Fanuc TP program (LS listing): S107_PK_T13N70.LS

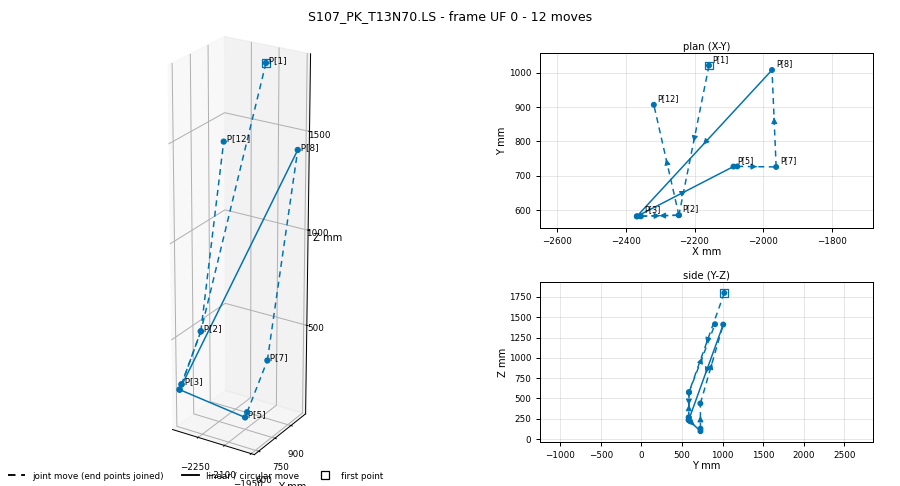
[picture p0: tool path of S107_PK_T13N70.LS in frame UF 0, 12 of 12 moves have a stored position in this frame; points joined in program order, loops and branches not executed]
/PROG  S107_PK_T13N70
/ATTR
OWNER		= MNEDITOR;
COMMENT		= "TL PCK TYP1 N70";
PROG_SIZE	= 4376;
CREATE		= DATE 21-06-09  TIME 09:54:06;
MODIFIED	= DATE 21-06-09  TIME 12:46:12;
FILE_NAME	= S107_PK_;
VERSION		= 0;
LINE_COUNT	= 155;
MEMORY_SIZE	= 4796;
PROTECT		= READ_WRITE;
STORAGE		= SHADOW;
TCD:  STACK_SIZE	= 0,
      TASK_PRIORITY	= 50,
      TIME_SLICE	= 0,
      BUSY_LAMP_OFF	= 0,
      ABORT_REQUEST	= 0,
      PAUSE_REQUEST	= 0;
DEFAULT_GROUP	= 1,*,*,*,*;
CONTROL_CODE	= 00000000 00000000;
/APPL
  HANDLING : TRUE ;
/MN
   1:  !******************************** ;
   2:  ! PATH - PK TOOL FROM N3=STA 70 ;
   3:  !******************************** ;
   4:  !* Robot ID: XXXXXR02B1 ;
   5:  !*    F-19XXXX ;
   6:  !* Line: XXXXXXXX ;
   7:  !* Platform: XX ;
   8:  !* Tool ID: TOOL xx ;
   9:  !* Program: S002_PK_TxxN3_R02 ;
  10:  !* Application: TOOL PICK ;
  11:  !******************************** ;
  12:  ! Author- Esys Automation ;
  13:  !******************************** ;
  14:   ;
  15:  !++++++++++++++++++++++++++++++++ ;
  16:  !ASSIGN PROGRAM PATH VALUES ;
  17:  !-------------------------------- ;
  18:  !Set ATI Tool and World UFrame ;
  19:  UTOOL_NUM=14 ;
  20:  UFRAME_NUM=0 ;
  21:  !++++++++++++++++++++++++++++++++ ;
  22:   ;
  23:  !******************************** ;
  24:  !BEGINNING OF PROGRAM PATH ;
  25:  !MOVE TO NEST 3 TOOL PICK ;
  26:  !******************************** ;
  27:   ;
  28:  !-------------------------------- ;
  29:  LBL[10:MOVE TO TL PICK] ;
  30:   ;
  31:  SET SEGMENT(52) ;
  32:  !SEG(52), Approach Tool Pick ;
  33:   ;
  34:J P[1] 100% CNT100    ;
  35:J P[2] 100% CNT100    ;
  36:J P[3] 100% CNT100    ;
  37:   ;
  38:L P[4:Pick Tool] 50mm/sec FINE    ;
  39:   ;
  40:  !-------------------------------- ;
  41:  LBL[20:LATCH TOOL] ;
  42:  LATCH TOOL    ;
  43:   ;
  44:  Set MH Tool(4) ;
  45:  Release Part(5) ;
  46:  VACUUM CAN 1 OFF(6,7) ;
  47:   ;
  48:  !Add MH Ethernet Device from ;
  49:  !I/O Ethernet table ;
  50:  !which tool has ;
  51:   ;
  52:  !ADD DEVICE ONLINE CALLS ;
  53:  !WITHOUT STATUS CHECK ARG ;
  54:  !FOR ALL EOAT DEVICES ;
  55:  !CALL EN_ONLN(x,y) ;
  56:  !x = EOAT ENET Node # ;
  57:  !y = wait time ;
  58:  CALL EN_ONLN(31,5) ;
  59:  CALL EN_AROFF(31) ;
  60:   ;
  61:  !If TL LCH Pass, Return Home ;
  62:  !If TL LCH Fail, Unlatch TL, ;
  63:  !  MHFault, and Return Home ;
  64:  IF R[170]=1,JMP LBL[30] ;
  65:   ;
  66:  SELECT R[168]=6,JMP LBL[80] ;
  67:         ELSE,JMP LBL[99] ;
  68:   ;
  69:  !-------------------------------- ;
  70:  LBL[30:TOOL CHECK] ;
  71:   ;
  72:  ! Check if Tool Match with PLC ;
  73:  CALL TL_CHK_KM(R[156]) ;
  74:   ;
  75:  !If TL CHK Pass, Return Home ;
  76:  !If TL CHK Fail, Unlatch Tool, ;
  77:  !  MHFault, and Return Home ;
  78:  IF R[170]=1,JMP LBL[40] ;
  79:  IF R[170]=0,JMP LBL[905] ;
  80:   ;
  81:  !-------------------------------- ;
  82:  LBL[40:COMPLETE PATH] ;
  83:  !TL PK COMPLETE. MOVE AWAY ;
  84:  !AND RETURN HOME ;
  85:   ;
  86:  !Set New Tool and World Frame ;
  87:  UTOOL_NUM=2 ;
  88:  UFRAME_NUM=0 ;
  89:   ;
  90:  !Set Payload= Tool ;
  91:  R[221]=2    ;
  92:  PAYLOAD[R[221]] ;
  93:   ;
  94:  SET SEGMENT(53) ;
  95:  !SEG(53), Tool Pick Depart ;
  96:   ;
  97:L P[5] 50mm/sec FINE    ;
  98:   ;
  99:L P[6] 1000mm/sec CNT100    ;
 100:J P[7] 100% CNT100    ;
 101:J P[8] 100% CNT100    ;
 102:   ;
 103:   ;
 104:  ! Move To Home ;
 105:  JMP LBL[100] ;
 106:   ;
 107:  !-------------------------------- ;
 108:  LBL[80:LATCHING FAULT] ;
 109:  !MOVE BACK TO HOME WITHOUT TOOL ;
 110:  !on Reverse Path before Tool Pick ;
 111:   ;
 112:  UNLATCH TOOL    ;
 113:   ;
 114:  UFRAME_NUM=0 ;
 115:  UTOOL_NUM=14 ;
 116:   ;
 117:L P[9] 50mm/sec FINE    ;
 118:   ;
 119:L P[10] 1000mm/sec CNT100    ;
 120:J P[11] 100% CNT100    ;
 121:J P[12] 100% CNT100    ;
 122:   ;
 123:   ;
 124:  SET SEGMENT(63) ;
 125:  !SEG(63), Robot Move to Home ;
 126:   ;
 127:  R[132]=0    ;
 128:  GO[71]=0 ;
 129:   ;
 130:  ! Move To Home ;
 131:  JMP LBL[100] ;
 132:   ;
 133:  !-------------------------------- ;
 134:  LBL[99:ABORT PROGRAM] ;
 135:  MESSAGE[...] ;
 136:  MESSAGE[ABORT PROGRAM] ;
 137:  ABORT ;
 138:   ;
 139:  !-------------------------------- ;
 140:  LBL[100:END OF PROGRAM] ;
 141:  END ;
 142:   ;
 143:  !***********FAULTS*********** ;
 144:  LBL[905:Invalid Tool Num] ;
 145:  MESSAGE[...] ;
 146:  MESSAGE[TOOL CHANGER FAULT] ;
 147:  MESSAGE[ ROBOT LATCHED TO] ;
 148:  MESSAGE[ WRONG TOOL.] ;
 149:  MESSAGE[ GI[70] DOES NOT ] ;
 150:  MESSAGE[ MATCH TOOL ID ] ;
 151:  DO[523]=ON ;
 152:  UALM[3] ;
 153:  DO[523]=OFF ;
 154:  JMP LBL[80] ;
 155:   ;
/POS
P[1]{
   GP1:
	UF : 0, UT : 14,		CONFIG : 'N U T, 0, 0, 0',
	X = -2157.965  mm,	Y =  1020.774  mm,	Z =  1799.157  mm,
	W =  -148.691 deg,	P =     -.556 deg,	R =    64.095 deg
};
P[2]{
   GP1:
	UF : 0, UT : 14,		CONFIG : 'N U T, 0, 0, 0',
	X = -2245.406  mm,	Y =   585.737  mm,	Z =   576.045  mm,
	W =  -160.449 deg,	P =      .486 deg,	R =    90.889 deg
};
P[3]{
   GP1:
	UF : 0, UT : 14,		CONFIG : 'N U T, 0, 0, 0',
	X = -2356.425  mm,	Y =   582.838  mm,	Z =   265.364  mm,
	W =  -160.444 deg,	P =      .210 deg,	R =    91.666 deg
};
P[4:"Pick Tool"]{
   GP1:
	UF : 0, UT : 14,		CONFIG : 'N U T, 0, 0, 0',
	X = -2367.590  mm,	Y =   582.398  mm,	Z =   233.916  mm,
	W =  -160.444 deg,	P =      .209 deg,	R =    91.666 deg
};
P[5]{
   GP1:
	UF : 0, UT : 2,		CONFIG : 'N U T, 0, 0, 0',
	X = -2086.858  mm,	Y =   727.136  mm,	Z =    96.569  mm,
	W =  -161.991 deg,	P =      .564 deg,	R =    90.288 deg
};
P[6]{
   GP1:
	UF : 0, UT : 2,		CONFIG : 'N U T, 0, 0, 0',
	X = -2075.694  mm,	Y =   727.576  mm,	Z =   128.016  mm,
	W =  -161.991 deg,	P =      .564 deg,	R =    90.288 deg
};
P[7]{
   GP1:
	UF : 0, UT : 2,		CONFIG : 'N U T, 0, 0, 0',
	X = -1962.717  mm,	Y =   725.991  mm,	Z =   438.063  mm,
	W =  -162.002 deg,	P =      .840 deg,	R =    89.511 deg
};
P[8]{
   GP1:
	UF : 0, UT : 2,		CONFIG : 'N U T, 0, 0, 0',
	X = -1974.745  mm,	Y =  1007.769  mm,	Z =  1410.068  mm,
	W =  -152.887 deg,	P =     -.534 deg,	R =    69.095 deg
};
P[9]{
   GP1:
	UF : 0, UT : 14,		CONFIG : 'N U T, 0, 0, 0',
	X = -2367.590  mm,	Y =   582.398  mm,	Z =   233.916  mm,
	W =  -160.444 deg,	P =      .209 deg,	R =    91.666 deg
};
P[10]{
   GP1:
	UF : 0, UT : 14,		CONFIG : 'N U T, 0, 0, 0',
	X = -2356.425  mm,	Y =   582.838  mm,	Z =   265.364  mm,
	W =  -160.444 deg,	P =      .210 deg,	R =    91.666 deg
};
P[11]{
   GP1:
	UF : 0, UT : 14,		CONFIG : 'N U T, 0, 0, 0',
	X = -2245.406  mm,	Y =   585.737  mm,	Z =   576.045  mm,
	W =  -160.449 deg,	P =      .486 deg,	R =    90.889 deg
};
P[12]{
   GP1:
	UF : 0, UT : 14,		CONFIG : 'N U T, 0, 0, 0',
	X = -2318.251  mm,	Y =   906.629  mm,	Z =  1414.240  mm,
	W =  -153.258 deg,	P =    -1.159 deg,	R =    74.791 deg
};
/END
